TYPE CoverPanelSetProcesses :
STRUCT
	///Reset any errors
	reset: Process;
END_STRUCT
END_TYPE

(* stored: Version 1.1.0.1, ProductVersion 3.1.4019.2
   DUT CoverPanelSetProcesses: Id {e2279cca-effb-435a-9917-d85fbb7ec056} *)
